FUNCTION_BLOCK insertLoadStation EXTENDS stateMachine
VAR_INPUT
	
	ioImage                : inserterLoadImage;

END_VAR

VAR

	activeState            : inserterLoadStates;	
	axisLinMot             : FB_ServoAxis_LinMot; 
	
	resetDone			   : BOOL := FALSE; 						   // Инсъртъра е ресетнат
	prepareStart           : BOOL := FALSE; 						   // Изчаква синхронизация с индекс масата
	loadStart              : BOOL := FALSE; 						   // Робота е донесъл нов сензор
	rotStart               : BOOL := FALSE; 						   // Начално поз. на ротатора
	posStart               : BOOL := FALSE; 						   // Ротира сензора на позиция, спрямо команда от камерата
	insertStart            : BOOL := FALSE;							   // Поставяне на сензора в гнездото на масата
	releaseStart           : BOOL := FALSE; 						   // Връщане на инсъртъра в начлана поз.
	syncStart			   : BOOL := FALSE; 						   // Sync с индекс масата, че работа е завършена

	
	initRotPos			   : REAL; 									   // Начално завъртане
	camRotPos              : REAL;                                     // Завъртане за снимка
	workRotPos             : REAL;                                     // Завъртане след снимка - cw ии ccw
	cwRotPos               : REAL;
    ccwRotPos              : REAL;     
	beforeGripPos          : REAL;                                 
	
	gripTime			   : TIME := T#350MS;                          // Време за ход на грипера
	gripTimeOut            : TIME := T#2S;                             // Време за отваряне/затваряне на гриперите
	insertTimeOut          : TIME := T#3S;                             // Време за движене нагоре/надолу на inserter 
    driveMoveTimeOut	   : TIME := T#4S;                             // Време за ход на мотора
	driveHomeTimeOut       : TIME := T#10S;                            // Време за home на мотора
	camTimeOut             : TIME := T#2S; 							   // Време за 1 снимка от камерата
	driveEnTime            : TIME := T#1S;                             // Време за ресет на инвертора на мотора
	drivePosTime           : TIME := T#100MS;                          // Време за задаване на задание за позициониране	

END_VAR


drivesControl();          // Упр. на ЛинМот мотора 

setStateVars(ioImage, activeState);


CASE activeState OF


//  *** Start Up
//  Старт на станцията след подаване на захр.	

	inserterLoadStates.stStartUp:
		setDisplayState(inserterLoadDisplayStates.dStStartUp);
		Stations.insertLoadDrive.DoEnable   := FALSE;
		Stations.insertLoadDrive.DoMove     := FALSE;	
		Stations.insertLoadDrive.DoHome     := FALSE;					   						   
		nextState(inserterLoadStates.stPowerUp);

//  *** Power Up - Start
//  Инициализация след подaване на захранване

	inserterLoadStates.stPowerUp:
		//IF io.getSR(ioImage.xGrip_close, ioImage.xGrip_open) THEN
			setError(inserterLoadStates.stErrInitSensor);
	//	END_IF
		nextState(inserterLoadStates.stInit);

//  *** Init 
//  Инициализация на станцията
	
	inserterLoadStates.stInit:
	
		depWait(globalDeps.depILoadInitDone);		
		
		IF NOT resetDone THEN
			nextState(inserterLoadStates.stResetStart);
		END_IF
		
		IF prepareStart THEN
			nextState(inserterLoadStates.stPrepareStart);
		END_IF
		
		IF loadStart THEN
			nextState(inserterLoadStates.stLoadStart);
		END_IF		
		
		IF rotStart THEN
			nextState(inserterLoadStates.stRotStart);
		END_IF

		IF posStart THEN
			nextState(inserterLoadStates.stPosStart);
		END_IF

		IF insertStart THEN
			nextState(inserterLoadStates.stInsertStart);		
		END_IF	

		IF releaseStart THEN
			nextState(inserterLoadStates.stReleaseStart);
		END_IF	

		IF syncStart THEN
			nextState(inserterLoadStates.stSyncIndexStart);
		END_IF		
			
		nextState(inserterLoadStates.stInitDone);
		
// *** Init Done

	inserterLoadStates.stInitDone:
		nextState(inserterLoadStates.stReady);
	
// *** Ready

	inserterLoadStates.stReady:	
		setDisplayState(inserterLoadDisplayStates.dStStandBy);	
		IF Global.purgeDoneIL THEN
			resetDone          := FALSE;		
			Global.purgeDoneIL := FALSE;
		END_IF
		depNextState(Stations.machineStBase, GlobalDeps.depMachineStopping,  inserterLoadStates.stInserterLoadStopped);
		depNextState(Stations.machineStBase, GlobalDeps.depMachineStop,      inserterLoadStates.stInserterLoadStopped);	
		depWait(globalDeps.depILoadWaitIndex);
		nextState(inserterLoadStates.stPrepareStart);

// *** Inserter is Stopped

	inserterLoadStates.stInserterLoadStopped:
		setDisplayState(inserterLoadDisplayStates.dStStationIsStopped);	
		depWait(globalDeps.depILoadStop);
		depNextState(stations.machineStBase, GlobalDeps.depMachineAuto,       inserterLoadStates.stReady);
	    depNextState(Stations.machineStBase, GlobalDeps.depMachinePurgeStart, inserterLoadStates.stReady);			
		Stations.insertLoadDrive.DoEnable   := FALSE;
		Stations.insertLoadDrive.DoMove     := FALSE;	
		Stations.insertLoadDrive.DoHome     := FALSE;		

// *** Reset - Start
// Ресетиране на inserter

	inserterLoadStates.stResetStart:
		setDisplayState(inserterLoadDisplayStates.dStStationIsReseting);		
		resetDone := FALSE;		
		nextState(inserterLoadStates.stResetSyncRobot);
		
// *** Reset - Robot Sync
// Робота трябва да е на безопастно растояние

	inserterLoadStates.stResetSyncRobot:
		IF NOT GLobal.robotSafe THEN	
			depWait(globalDeps.depILoadWaitRobotReady);
			nextState(inserterLoadStates.stResetGripOpen);	
		ELSE
			nextState(inserterLoadStates.stResetGripOpen);	
		END_IF			

// *** Reset - Grip Open
// Отваряне на грипера

	inserterLoadStates.stResetGripOpen:
		io.setSR(ioImage.yGrip_open, ioImage.yGrip_close);
		nextState(inserterLoadStates.stResetGripCheck);	

// *** Reset - Grip Check
// Проверка дали грипера се е отворил
// Движение на гора на инсертъра

	inserterLoadStates.stResetGripCheck:		
 		IF io.getSR(ioImage.xGrip_open, ioImage.xGrip_close) THEN
			io.setSR(ioImage.yInsert_up, ioImage.yInsert_down);
			nextState(inserterLoadStates.stResetMoveUpCheck);	
		END_IF
		timeOutError(gripTimeOut, inserterLoadStates.stErrGripNotOpen);
		
// *** Reset - Move Up Check
// Проверка дали инсертъра е горе

	inserterLoadStates.stResetMoveUpCheck:		
		IF io.getSR(ioImage.xInsert_up, ioImage.xInsert_down) THEN
			nextState(inserterLoadStates.stResetLimitsCalc);			
		END_IF
		timeOutError(insertTimeOut, inserterLoadStates.stErrInsertNotUp);	
			
// *** Reset - Limit Check
// В зависимост от избраният модел на продукт се зараждат настойки в инвертора на мотора

	inserterLoadStates.stResetLimitsCalc:
			
		initRotPos    := Stations.insertLoadSetting.rotParams[Global.recipe].initRot;
		camRotPos     := Stations.insertLoadSetting.rotParams[Global.recipe].camRot;
		beforeGripPos := Stations.insertLoadSetting.rotParams[Global.recipe].beforeGripRot;
		cwRotPos      := Stations.insertLoadSetting.rotParams[Global.recipe].cwRot;
		ccwRotPos     := Stations.insertLoadSetting.rotParams[Global.recipe].ccwRot;
		
		IF Stations.insertLoadDrive.Error THEN
			Stations.insertLoadDrive.DoReset  := TRUE;
		ELSE
			Stations.insertLoadDrive.DoReset  := FALSE;
			Stations.insertLoadDrive.DoEnable := TRUE;
			IF stateDelay(driveEnTime) THEN
				nextState(inserterLoadStates.stResetDriveHome);
			END_IF
		END_IF
		timeOutError(driveEnTime*2, inserterLoadStates.stErrDriveErr);
		
// *** Reset - Drive Home
// Рефериране на мотора

	inserterLoadStates.stResetDriveHome:		
		IF Stations.insertLoadDrive.Enabled AND NOT Stations.insertLoadDrive.Error THEN	
			Stations.insertLoadDrive.DoHome := TRUE;
			IF stateDelay(driveEnTime) THEN
				nextState(inserterLoadStates.stResetDriveCheck1);	
			END_IF
		ELSE
			setError(inserterLoadStates.stErrDriveErr);
	   END_IF	
		
// *** Reset - Drive Check
// Проверка дали реферирането на мотора е завършено

	inserterLoadStates.stResetDriveCheck1:		
		IF Stations.insertLoadDrive.Refferenced AND NOT Stations.insertLoadDrive.Error THEN
			Stations.insertLoadDrive.DoHome := FALSE;
			nextState(inserterLoadStates.stResetDriveMove);	
		END_IF
		timeOutError(driveHomeTimeOut, inserterLoadStates.stErrDriveHome);	

// *** Reset - Drive Move
// Ротатора застава на начална позиция

	inserterLoadStates.stResetDriveMove:
		IF Stations.insertLoadDrive.Enabled AND NOT Stations.insertLoadDrive.Error THEN	
			Stations.insertLoadDrive.TargetVelocity      := Stations.insertLoadSetting.axisWorkSpeed;
			Stations.insertLoadDrive.TargetAcceleration  := Stations.insertLoadSetting.axisAcc;
			Stations.insertLoadDrive.TargetPrecision     := Stations.insertLoadSetting.axisPres;
			Stations.insertLoadDrive.TargetPosition      := initRotPos;
		    Stations.insertLoadDrive.DoMove              := TRUE;
			IF stateDelay(driveEnTime) THEN			
				nextState(inserterLoadStates.stResetDriveCheck2);	
			END_IF
		ELSE
			setError(inserterLoadStates.stErrDriveErr);
	   END_IF	
	   
// *** Reset - Drive Check2
// Проверка дали реферирането на мотора е завършено

	inserterLoadStates.stResetDriveCheck2:		
		IF Stations.insertLoadDrive.TargetReached AND NOT Stations.insertLoadDrive.Error THEN
			Stations.insertLoadDrive.DoMove := FALSE;
			nextState(inserterLoadStates.stResetDone);	
		ELSIF NOT Stations.insertLoadDrive.TargetReached AND Stations.insertLoadDrive.Error THEN
			setError(inserterLoadStates.stErrDriveErr);
		END_IF	
		timeOutError(driveMoveTimeOut, inserterLoadStates.stErrDriveTimeOut);	

// *** Reset - Done

	inserterLoadStates.stResetDone:		
		resetDone := TRUE;
	    nextState(inserterLoadStates.stReady);			
		
// *** Prepare - Start
// Индекс масата е завършила ходата си - чака се робота да донесе сензор

	inserterLoadStates.stPrepareStart:
	   setDisplayState(inserterLoadDisplayStates.dStWorking);
	   prepareStart := TRUE;
	   nextState(inserterLoadStates.stPrepareNestCheck);	   
	   
// *** Prepare - Nest Check
// Ако в масата има зареден сенсор - станцията преключва работа
// Иначе дава сигнал на робота, че очаква от него да донесе сензор

	inserterLoadStates.stPrepareNestCheck:	   
		IF NOT io.getX(ioImage.xNest) AND NOT Global.purgeActive THEN
 	       nextState(inserterLoadStates.stPrepareRobotWait);  
        ELSE
	        prepareStart := FALSE;
 	        nextState(inserterLoadStates.stSyncIndexStart);  			
        END_IF	
	  
// *** Prepare - Robot Wait
// Изчаква робота да донесе сензор 

	inserterLoadStates.stPrepareRobotWait:		
		depSignal(globalDeps.depILoadSignalForLoad);
		depNextState(Stations.roboStBase, globalDeps.depRoboILoadOnPos, inserterLoadStates.stPrepareDone);
	
// *** Prepare - Done 

	inserterLoadStates.stPrepareDone:		
		prepareStart    := FALSE;
		nextState(inserterLoadStates.stLoadStart);
		
// *** Load - Start
// Сензора трябва да се прехвърли от робота в грипера на инсъртъра
		
	inserterLoadStates.stLoadStart:			
		loadStart   := TRUE;
		IF Stations.insertLoadDrive.Enabled AND NOT Stations.insertLoadDrive.Error THEN
			nextState(inserterLoadStates.stLoadDriveMove);	
		ELSE
			nextState(inserterLoadStates.stLoadDriveOn);			
		END_IF	
		
// *** Load - Drive On
// Ако е затворен грипера, пуска мотора 	
		
	inserterLoadStates.stLoadDriveOn:
		IF Stations.insertLoadDrive.Error THEN
			Stations.insertLoadDrive.DoReset  := TRUE;
		ELSE
			Stations.insertLoadDrive.DoReset  := FALSE;
			Stations.insertLoadDrive.DoEnable := TRUE;
			IF stateDelay(driveEnTime) THEN
				nextState(inserterLoadStates.stLoadDriveMove);
			END_IF
		END_IF
		timeOutError(driveEnTime*2, inserterLoadStates.stErrDriveErr);
		
// *** Pos - Drive Move
// Завърта мотора	

	inserterLoadStates.stLoadDriveMove:
		IF Stations.insertLoadDrive.Enabled AND NOT Stations.insertLoadDrive.Error THEN	
			Stations.insertLoadDrive.TargetVelocity      := Stations.insertLoadSetting.axisWorkSpeed;
			Stations.insertLoadDrive.TargetAcceleration  := Stations.insertLoadSetting.axisAcc;
			Stations.insertLoadDrive.TargetPrecision     := Stations.insertLoadSetting.axisPres;
			Stations.insertLoadDrive.TargetPosition      := beforeGripPos;
		    Stations.insertLoadDrive.DoMove              := TRUE;
			IF stateDelay(driveEnTime) THEN			
				nextState(inserterLoadStates.stLoadDriveCheck);	
			END_IF
		ELSE
			setError(inserterLoadStates.stErrDriveErr);
	   END_IF	

// *** Load - Drive Check
// Проверка дали мотора си е завършил хода

	inserterLoadStates.stLoadDriveCheck:
		IF Stations.insertLoadDrive.TargetReached AND NOT Stations.insertLoadDrive.Error THEN
			Stations.insertLoadDrive.DoMove := FALSE;
			io.setSR(ioImage.yGrip_close, ioImage.yGrip_open);
			IF stateDelay(gripTime) THEN
				nextState(inserterLoadStates.stLoadGripCheck);	
			END_IF
		ELSIF NOT Stations.insertLoadDrive.TargetReached AND Stations.insertLoadDrive.Error THEN
			setError(inserterLoadStates.stErrDriveErr);
		END_IF	
		timeOutError(driveMoveTimeOut, inserterLoadStates.stErrDriveTimeOut);	
		
// *** Load - Gripper Check
// Проверява се дали се е затворил грипера на инсъртъра

	inserterLoadStates.stLoadGripCheck:	
		// За сега не може да се настрой сензора на затворено пол. - затова е заместен с чисто закъснение	
		// IF io.getSR(ioImage.xGrip_close, ioImage.xGrip_open) THEN
			nextState(inserterLoadStates.stLoadRobotSync);	
		// END_IF	
		// timeOutError(gripTimeOut, inserterLoadStates.stErrGripNotClose);		
		
// *** Load - Robo Sync
// Дава се сигнал робота да си отвори грипера

	inserterLoadStates.stLoadRobotSync:			
		depWait(globalDeps.depRoboGripOpen);
		depNextState(Stations.roboStBase, GlobalDeps.depILoadRobotBack, inserterLoadStates.stLoadDone);

// *** Load - Done

	inserterLoadStates.stLoadDone:			
		loadStart  := FALSE;
		nextState(inserterLoadStates.stRotStart);		

// *** Rot - Start
// Започва ротиране на сензора, за да може да бъде сниман

	inserterLoadStates.stRotStart:	
		rotStart    := TRUE;
		io.setSR(ioImage.yGrip_close, ioImage.yGrip_open);
		nextState(inserterLoadStates.stRotGripCheck);

// *** Rot - Grip Check
// Ако е затворен грипера, пуска мотора 

	inserterLoadStates.stRotGripCheck:
		// За сега не може да се настрой сензора на затворено пол. 
		IF Stations.insertLoadDrive.Enabled AND NOT Stations.insertLoadDrive.Error THEN
			nextState(inserterLoadStates.stRotDriveMove);	
		ELSE
			nextState(inserterLoadStates.stRotDriveOn);			
		END_IF
		timeOutError(gripTimeOut, inserterLoadStates.stErrGripNotClose);
		
// *** Rot - Drive On
// Ако е затворен грипера, пуска мотора 

	inserterLoadStates.stRotDriveOn:
		IF Stations.insertLoadDrive.Error THEN
			Stations.insertLoadDrive.DoReset  := TRUE;
		ELSE
			Stations.insertLoadDrive.DoReset  := FALSE;
			Stations.insertLoadDrive.DoEnable := TRUE;
			IF stateDelay(driveEnTime) THEN
				nextState(inserterLoadStates.stRotDriveMove);
			END_IF
		END_IF
		timeOutError(driveEnTime*2, inserterLoadStates.stErrDriveErr);

// *** Rot - Drive Move
// Завърта мотора на поз. за снимане

	inserterLoadStates.stRotDriveMove:
		IF Stations.insertLoadDrive.Enabled AND NOT Stations.insertLoadDrive.Error THEN	
			Stations.insertLoadDrive.TargetVelocity      := Stations.insertLoadSetting.axisWorkSpeed;
			Stations.insertLoadDrive.TargetAcceleration  := Stations.insertLoadSetting.axisAcc;
			Stations.insertLoadDrive.TargetPrecision     := Stations.insertLoadSetting.axisPres;
			Stations.insertLoadDrive.TargetPosition      := camRotPos;
		    Stations.insertLoadDrive.DoMove              := TRUE;	
			IF stateDelay(driveEnTime) THEN		
				nextState(inserterLoadStates.stRotDriveCheck);	
			END_IF
		ELSE
			setError(inserterLoadStates.stErrDriveErr);
	   END_IF	

// *** Rot - Drive Check
// Проверка дали мотора си е завършил хода

	inserterLoadStates.stRotDriveCheck:
		IF Stations.insertLoadDrive.TargetReached AND NOT Stations.insertLoadDrive.Error THEN
			Stations.insertLoadDrive.DoMove := FALSE;
			io.setY(ioImage.yFlashLight);
			nextState(inserterLoadStates.stRotCamShot);	
		ELSIF NOT Stations.insertLoadDrive.TargetReached AND Stations.insertLoadDrive.Error THEN
			setError(inserterLoadStates.stErrDriveErr);
		END_IF	
		timeOutError(driveMoveTimeOut, inserterLoadStates.stErrDriveTimeOut);

// *** Rot - Cam Shot
// Прави се снимка на сензора

	inserterLoadStates.stRotCamShot:
		Stations.insertLoadData := Global.recipe;
		nextState(inserterLoadStates.stRotCamCheck);

// *** Rot - Cam Check
// Проверява се дали има успешна снимка и върнат резултат

	inserterLoadStates.stRotCamCheck:
		IF Stations.insertLoadData = dataRequestCam.done THEN 
			
			IF TagsHMI.camResult <> camResult.null THEN
				
				CASE TagsHMI.camResult OF 
						camResult.turnCCW : workRotPos := camRotPos + ccwRotPos;
						camResult.turnCW  : workRotPos := camRotPos + cwRotPos;
				END_CASE
				nextState(inserterLoadStates.stRotDone);
				
			ELSE
				setError(inserterLoadStates.stErrCamBadResult);				
			END_IF
		
		ELSIF Stations.insertLoadData = dataRequestCam.error THEN
			setError(inserterLoadStates.stErrCamErr);			
		END_IF
		io.rstY(ioImage.yFlashLight);
		timeOutError(camTimeOut, inserterLoadStates.stErrCamTimeout);		
		
// *** Rot - Done

	inserterLoadStates.stRotDone:		
		rotStart   := FALSE;
		nextState(inserterLoadStates.stPosStart);		
		
// *** Pos  - Start
// Трябва да се завърти сензора на базата на резултата от камерата

	inserterLoadStates.stPosStart:		
		posStart   := TRUE;
		io.setSR(ioImage.yGrip_close, ioImage.yGrip_open);
		nextState(inserterLoadStates.stPosGripCheck);		
			
// *** Pos - Grip Check

	inserterLoadStates.stPosGripCheck:
		// За сега не може да се настрой сензора на затворено пол. - затова е заместен с чисто закъснение
		// IF io.getSR(ioImage.xGrip_close, ioImage.xGrip_open) THEN
		IF Stations.insertLoadDrive.Enabled AND NOT Stations.insertLoadDrive.Error THEN
			nextState(inserterLoadStates.stPosDriveMove);	
		ELSE
			nextState(inserterLoadStates.stPosDriveOn);			
		END_IF
		// END_IF	
		timeOutError(gripTimeOut, inserterLoadStates.stErrGripNotClose);	
		
// *** Pos - Drive On
// Ако е затворен грипера, пуска мотора 

	inserterLoadStates.stPosDriveOn:
		IF Stations.insertLoadDrive.Error THEN
			Stations.insertLoadDrive.DoReset  := TRUE;
		ELSE
			Stations.insertLoadDrive.DoReset  := FALSE;
			Stations.insertLoadDrive.DoEnable := TRUE;
			IF stateDelay(driveEnTime) THEN
				nextState(inserterLoadStates.stPosDriveMove);
			END_IF
		END_IF
		timeOutError(driveEnTime*2, inserterLoadStates.stErrDriveErr);	
		
// *** Pos - Drive Move
// Завърта мотора 

	inserterLoadStates.stPosDriveMove:
		IF Stations.insertLoadDrive.Enabled AND NOT Stations.insertLoadDrive.Error THEN	
			Stations.insertLoadDrive.TargetVelocity      := Stations.insertLoadSetting.axisWorkSpeed;
			Stations.insertLoadDrive.TargetAcceleration  := Stations.insertLoadSetting.axisAcc;
			Stations.insertLoadDrive.TargetPrecision     := Stations.insertLoadSetting.axisPres;
			Stations.insertLoadDrive.TargetPosition      := workRotPos;
		    Stations.insertLoadDrive.DoMove              := TRUE;
			IF stateDelay(driveEnTime) THEN			
				nextState(inserterLoadStates.stPosDriveCheck);	
			END_IF
		ELSE
			setError(inserterLoadStates.stErrDriveErr);
	   END_IF	
		
// *** Pos - Drive Check
// Проверка дали мотора си е завършил хода

	inserterLoadStates.stPosDriveCheck:
		IF Stations.insertLoadDrive.TargetReached AND NOT Stations.insertLoadDrive.Error THEN
			Stations.insertLoadDrive.DoMove := FALSE;
			nextState(inserterLoadStates.stPosDone);	
		ELSIF NOT Stations.insertLoadDrive.TargetReached AND Stations.insertLoadDrive.Error THEN
			setError(inserterLoadStates.stErrDriveErr);
		END_IF	
		timeOutError(driveMoveTimeOut, inserterLoadStates.stErrDriveTimeOut);			   
	   
// *** Pos - Done

	inserterLoadStates.stPosDone:
		posStart   := FALSE;
		nextState(inserterLoadStates.stInsertStart);	  

// *** Insert - Start
// Поставя сензора на в гнездото на индекс масата

	inserterLoadStates.stInsertStart:
		insertStart := TRUE;
		io.setSR(ioImage.yGrip_close, ioImage.yGrip_open);
		nextState(inserterLoadStates.stInsertGripCheck);	

// *** Insert - Grip Check
// Проверява се дали грипера е затворен

	inserterLoadStates.stInsertGripCheck:
	// За сега не може да се настрой сензора на затворено пол.
		//IF io.getSR(ioImage.xGrip_close, ioImage.xGrip_open) THEN
			nextState(inserterLoadStates.stInsertNestCheck);		
		//END_IF
		timeOutError(gripTimeOut, inserterLoadStates.stErrGripNotClose);
		
// *** Insert - Nest Check
// Сензор се поставя само ако на масата няма

	inserterLoadStates.stInsertNestCheck:
		IF NOT io.getX(ioImage.xNest) THEN
			io.setSR(ioImage.yInsert_down, ioImage.yInsert_up);
			nextState(inserterLoadStates.stInsertMoveDownCheck);			
		ELSE
			setError(inserterLoadStates.stErrInitSensor);
		END_IF
		
// *** Insert - Insert Move Down Check
// Проверява се дали е инсъртъра е долу

	inserterLoadStates.stInsertMoveDownCheck:		
		IF io.getSR(ioImage.xInsert_down, ioImage.xInsert_up) THEN
			nextState(inserterLoadStates.stInsetDone);			
		END_IF	
		timeOutError(insertTimeOut, inserterLoadStates.stErrInsertNotDown);

// *** Insert - Done

	inserterLoadStates.stInsetDone:	 
		insertStart := FALSE;
		nextState(inserterLoadStates.stReleaseStart);		
	   
// *** Release - Start
// Оставяне на сензора в гнездота и връщата в начална поз.

	inserterLoadStates.stReleaseStart:	   
		releaseStart := TRUE;
		io.setSR(ioImage.yGrip_open, ioImage.yGrip_close);
		nextState(inserterLoadStates.stReleaseGripCheck);	

// *** Release - Grip Check
// Проверка дали грипера се е отворил

	inserterLoadStates.stReleaseGripCheck:	   
		IF io.getSR(ioImage.xGrip_open, ioImage.xGrip_close) THEN
			io.setSR(ioImage.yInsert_up, ioImage.yInsert_down);
			nextState(inserterLoadStates.stReleaseMoveUpCheck);			
		END_IF	
		timeOutError(gripTimeOut, inserterLoadStates.stErrGripNotOpen);				   
	
// *** Release - Move Up Check
// Проверка дали инсъртъра е горе

	inserterLoadStates.stReleaseMoveUpCheck:
		IF io.getSR(ioImage.xInsert_up, ioImage.xInsert_down) THEN
			IF Stations.insertLoadDrive.Enabled AND NOT Stations.insertLoadDrive.Error THEN
				nextState(inserterLoadStates.stReleaseDriveMove);	
			ELSE
			    nextState(inserterLoadStates.stReleaseDriveOn);			
			END_IF			
		END_IF
		timeOutError(insertTimeOut, inserterLoadStates.stErrInsertNotUp);	

// *** Release - Drive On
// Ако инсъртъра е горе , пуска мотора 

	inserterLoadStates.stReleaseDriveOn:
		IF Stations.insertLoadDrive.Error THEN
			Stations.insertLoadDrive.DoReset  := TRUE;
		ELSE
			Stations.insertLoadDrive.DoReset  := FALSE;
			Stations.insertLoadDrive.DoEnable := TRUE;
			IF stateDelay(driveEnTime) THEN
				nextState(inserterLoadStates.stReleaseDriveMove);
			END_IF
		END_IF
		timeOutError(driveEnTime*2, inserterLoadStates.stErrDriveErr);	
		
// *** Release - Drive Move
// Завърта мотора 

	inserterLoadStates.stReleaseDriveMove:
		IF Stations.insertLoadDrive.Enabled AND NOT Stations.insertLoadDrive.Error THEN	
			Stations.insertLoadDrive.TargetVelocity      := Stations.insertLoadSetting.axisWorkSpeed;
			Stations.insertLoadDrive.TargetAcceleration  := Stations.insertLoadSetting.axisAcc;
			Stations.insertLoadDrive.TargetPrecision     := Stations.insertLoadSetting.axisPres;
			Stations.insertLoadDrive.TargetPosition      := initRotPos;
		    Stations.insertLoadDrive.DoMove              := TRUE;
			IF stateDelay(driveEnTime) THEN			
				nextState(inserterLoadStates.stReleaseDriveCheck);	
			END_IF
		ELSE
			setError(inserterLoadStates.stErrDriveErr);
	   END_IF	
		
// *** Release - Drive Check
// Проверка дали мотора си е завършил хода

	inserterLoadStates.stReleaseDriveCheck:
		IF Stations.insertLoadDrive.TargetReached AND NOT Stations.insertLoadDrive.Error THEN
			Stations.insertLoadDrive.DoMove := FALSE;
			nextState(inserterLoadStates.stReleaseDone);	
		ELSIF NOT Stations.insertLoadDrive.TargetReached AND Stations.insertLoadDrive.Error THEN
			setError(inserterLoadStates.stErrDriveErr);
		END_IF	
		timeOutError(driveMoveTimeOut, inserterLoadStates.stErrDriveTimeOut);  
	   
// *** Release - Done

	inserterLoadStates.stReleaseDone:	
        setDisplayState(inserterLoadDisplayStates.dStStationReady);	
		releaseStart  := FALSE;
		nextState(inserterLoadStates.stSyncIndexStart);

// *** Sync Index - Start
// Дава се разрешение да се завърти индекс масата

	inserterLoadStates.stSyncIndexStart:
		syncStart := TRUE;		
		depWait(globalDeps.depILoadDone);	
		depNextState(Stations.incCommStBase, globalDeps.depIncCycleDone, inserterLoadStates.stSyncIndexDone); 

// *** Sync Index - Done

	inserterLoadStates.stSyncIndexDone:
		syncStart := FALSE;
		nextState(inserterLoadStates.stReady);   
	        
// *** Step Block State
// В този state се влиза винаги след изпълняването на една стъпка при стъпков режим
	inserterLoadStates.stStepBlock:
        setDisplayState(inserterLoadDisplayStates.dStWaitForNextStep);	
		
// *** Station Stop
// Станцията е била изключена 
 
	inserterLoadStates.stStop: 	
		Stations.insertLoadDrive.DoEnable   := FALSE;
		Stations.insertLoadDrive.DoMove     := FALSE;	
	    resetDone			                := FALSE; 						   
	    prepareStart                        := FALSE; 						   
	    loadStart                           := FALSE; 						   
	    rotStart                            := FALSE; 						   
	    posStart                            := FALSE; 						   
	    insertStart                         := FALSE;							  
	    releaseStart                        := FALSE; 						   
	    syncStart			                := FALSE; 

// *** ERROR - Grip Not Open
// Грипера не се е отворил на време

	inserterLoadStates.stErrGripNotOpen:
		setDisplayState(inserterLoadDisplayStates.dStGripperDidNotOpen); 

// *** ERROR - Grip Not Close
// Грипера не се е затворил на време

	inserterLoadStates.stErrGripNotClose:
		setDisplayState(inserterLoadDisplayStates.dStGripperDidNotClose);
		
// *** ERROR - Inserter Not Down
// Inserter не е стинглал долна позиция на време

	inserterLoadStates.stErrInsertNotDown:
		setDisplayState(inserterLoadDisplayStates.dStInserterDidNotMoveDown);		
		
// *** ERROR - Inserter Not Up
// Inserter не е стинглал горна позиция на време

	inserterLoadStates.stErrInsertNotUp:
		setDisplayState(inserterLoadDisplayStates.dStInserterDidNotMoveUp);		
		
// *** ERROR - Drive Homming TimeOut
// ЛинМот мотора не е могъл да се homming както трябва

	inserterLoadStates.stErrDriveHome:
		setDisplayState(inserterLoadDisplayStates.dStDriveDidNotHome);
		Stations.insertLoadDrive.DoEnable   := FALSE;
		Stations.insertLoadDrive.DoMove     := FALSE;	
		Stations.insertLoadDrive.DoHome     := FALSE;	
		
// *** ERROR - Drive Homming TimeOut
// ЛинМот инвертора е върнал грешка

	inserterLoadStates.stErrDriveErr:
		setDisplayState(inserterLoadDisplayStates.dStDriveError);	
		Stations.insertLoadDrive.DoEnable   := FALSE;
		Stations.insertLoadDrive.DoMove     := FALSE;		
		
// *** ERROR - Drive Move TimeOut
// ЛинМот мотора не е завършил движението си навреме

	inserterLoadStates.stErrDriveTimeOut:
		setDisplayState(inserterLoadDisplayStates.dStDriveTimeOutMove);	
		Stations.insertLoadDrive.DoEnable   := FALSE;
		Stations.insertLoadDrive.DoMove     := FALSE;		
		
// *** ERROR - Camera Timeout
// Камерата се е забавила твърде мн. с връщането на резултат

	inserterLoadStates.stErrCamTimeout:
		setDisplayState(inserterLoadDisplayStates.dStCameraTimeOut);
		
// *** ERROR - Camera Error
// Камерата се е забавила твърде мн. с връщането на резултат

	inserterLoadStates.stErrCamErr:
		setDisplayState(inserterLoadDisplayStates.dStCameraError);
		
// *** ERROR - Camera Error
// Камерата е върнала грешен резултат

	inserterLoadStates.stErrCamBadResult:
		setDisplayState(inserterLoadDisplayStates.dStCameraBadResult);	
		
	
// *** ERROR - Init sensor 
// При старт на машаината не може да има захванат от грипера сензор

	inserterLoadStates.stErrInitSensor:	
		setDisplayState(inserterLoadDisplayStates.dStInitSensorGripError);	
		
// *** EMG Stop
// Аварийно спиране при натискане на гъба или отваряне на врата

	inserterLoadStates.stEMG:		
		Stations.insertLoadDrive.DoEnable   := FALSE;
		Stations.insertLoadDrive.DoMove     := FALSE;	
		Stations.insertLoadDrive.DoHome     := FALSE;
		nextState(inserterLoadStates.stInit);		


END_CASE

ACTION drivesControl:


axisLinMot       ( TargetPosition 		   := Stations.insertLoadDrive.TargetPosition,
				   TargetVelocity 		   := Stations.insertLoadDrive.TargetVelocity,
				   TargetAcceleration	   := Stations.insertLoadDrive.TargetAcceleration,
				   TargetDeceleration	   := Stations.insertLoadDrive.TargetAcceleration,
				   TargetPrecision 		   := Stations.insertLoadDrive.TargetPrecision,			
				   IsAbsolute 			   := FALSE,
	               OperationMode		   := Stations.insertLoadDrive.OperationMode,     				
	               Enabled 				   => Stations.insertLoadDrive.Enabled,
	               Error 				   => Stations.insertLoadDrive.Error,
	               ErrorID 				   => Stations.insertLoadDrive.ErrorID,
	               Refferenced 			   => Stations.insertLoadDrive.Refferenced,
	               Moving 				   => Stations.insertLoadDrive.Moving,
	               CurrentPosition 		   => Stations.insertLoadDrive.CurrentPosition,
	               CurrentVelocity		   => Stations.insertLoadDrive.CurrentVelocity,             				
				   Axis					   := Stations.insertLoadAxis,
		           DoServoOn 			   := Stations.insertLoadDrive.DoEnable, 
	               DoHome 				   := Stations.insertLoadDrive.DoHome, 
	               DoMove 				   := Stations.insertLoadDrive.DoMove, 
	               DoReset 				   := Stations.insertLoadDrive.DoReset, 
	               TargetReached 		   := Stations.insertLoadDrive.TargetReached, 
	               DoStop 				   := Stations.insertLoadDrive.DoStop);
END_ACTION

END_FUNCTION_BLOCK

(* stored: Version 1.1.0.1, ProductVersion 3.1.4024.3
   POU insertLoadStation: Id {6268782d-4abc-4a81-9966-96c42ef0fea5}, SpecialFunc None
   Action drivesControl: Id {a98c116b-c2d9-423d-a486-22093ca943a8} *)
